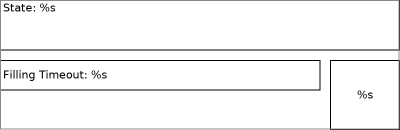
VISUALIZATION Vi_TankCtrl  // 400x130
VAR_IN_OUT
	hmi			: TankCtrl_Hmi;
END_VAR
    Rectangle (0,0 400x50), "State: %s", text variable: hmi.sStatusText
        p55702900: hmi.nStatusTextColor
    Rectangle (330,60 70x70), "%s", text variable: hmi.nMultiButtonText, invisible if: NOT hmi.bMultiButtonVis, colour variable: hmi.nMultiButtonColor
        toggle hmi.bMultiButton
    Rectangle (0,60 320x30), "Filling Timeout: %s", text variable: Strf.SimpleTime(UDINT_TO_TIME(hmi.nFillingTimeout.val * 1000), 'S', 'M')
        OnMouseUp: write hmi.nFillingTimeout.val via Default, min 0
END_VISUALIZATION

(* stored: Version 1.1.0.1
   Visu Vi_TankCtrl: Id {d92bdb92-07b5-488b-bd16-2022a6d5ab36} *)
